// TIA Portal V20 export
DATA_BLOCK "ET200SP_202"   // DB273
// stored: MemoryReserve 100
   VAR
      "SP202.00 AUTO INITIATE PBL LAMP ON (GREEN)" : Bool;
      "SP202.01 STOP PBL LAMP ON (RED)" : Bool;
      SPARE1 : Bool;
      "SP202.03 ENABLE PBL LAMP ON (BLACK)" : Bool;
      "SP202.04 SAFETY RESET PBL LAMP ON (BLUE)" : Bool;
      SPARE2 : Bool;
      SPARE3 : Bool;
      SPARE4 : Bool;
      "SP202.08 TOWER LAMP 1 ON (RED)" : Bool;
      "SP202.09 TOWER LAMP 2 ON (AMBER)" : Bool;
      "SP202.10 TOWER LAMP 3 ON (GREEN)" : Bool;
      "SP202.11 TOWER LAMP 4 ON (WHITE)" : Bool;
      "SP202.12 TOWER LAMP 5 ON (BLUE)" : Bool;
      "SP202.13 TOWER LAMP 6 ON (BUZZER)" : Bool;
      SPARE5 : Bool;
      SPARE6 : Bool;
   END_VAR
BEGIN
END_DATA_BLOCK
